// TIA Portal V16 export
// export: Created 2022-02-11T10:42:49.548867Z, ExportSetting WithDefaults, DisplayName Totally Integrated Automation Portal, DisplayVersion V16 Update 5, DisplayName TIA Portal Version Control Interface, DisplayVersion V16 Update 2, DisplayName TIA Portal Openness, DisplayVersion V16 Update 5, DisplayName STEP 7 Professional, DisplayVersion V16 Update 5, DisplayName STEP 7 Safety, DisplayVersion V16, DisplayName WinCC Professional, DisplayVersion V16 Update 5, DisplayName SIMATIC Visualization Architect, DisplayVersion V16
FUNCTION_BLOCK "fbObjEV_Aireacio"   // FB9102, LAD
{ S7_Optimized_Access := 'TRUE' }
VERSION : 0.1
// stored: AutoNumber false, IsIECCheckEnabled false, IsRetainMemResEnabled false, MemoryReserve 0, SetENOAutomatically false, UDAEnableTagReadback false
   VAR_INPUT
      eDP_PosTra : Bool := FALSE;   // Detector posicio valvula oberta
      eDP_PosAir : Bool := TRUE;   // Detector posicio valvula tancada
      aPosTra_Auto : Bool := FALSE;   // Ordre obrir EV en automatic
      psEnaAutoGrl : "boto";
      psEnaManualGrl : "boto";
      bCM_DirTra : Bool := TRUE;   // Condicions necesaries obrir valvula
      tAla_DirTra : Time := t#5s;   // Temps retard activacio alarma error obrir EV
      tAla_DirAir : Time := t#5s;   // Temps retard activacio alarma error tancar EV
      tAla_CM_DirTra : Time := t#3s;   // Temps retard activacio alarma condicions moviment
      psAnuConMov : Bool;
      psResetAlarma : Bool;
      mFirstScan : Bool;
      "Clock_0.5Hz" : Bool;
      bSysOk : Bool;
   END_VAR
   VAR_OUTPUT
      aPosTra : Bool;   // Sortida activacio EV
      be_DirTra : Bool;   // Bit estat EV oberta (Detectors + Sortida)
      be_DirAir : Bool;   // Bit estat EV tancada (Detectors + Sortida)
      al_CM_PosTra : Bool;   // Alarma condicions moviment obrir
      al_PosTra : Bool;   // Alarma obrir EV
      al_PosAir : Bool;   // Alarma tancar EV
      al_psEna : Bool;
   END_VAR
   VAR
      HMI { S7_SetPoint := 'True'} : "HMI_oEV";
      timAla_CM_DirTra : IEC_TIMER;   // Timer retard alarma condicions moviment
      timAla_DirTra : IEC_TIMER;   // Timer retard alarma obrirEV
      timAla_DirAir : IEC_TIMER;   // Timer retard alarma tancar EV
      mAuxTimer : Bool;   // Bit auxiliarInicialitzacio timers
      bLast_Reset : Bool;
   END_VAR
   VAR_TEMP
      ModeManual : Bool;
      ModeAutomatic : Bool;
      be_DirTra_Err : Bool;   // Error en validacio EV oberta. Sense retard per alarma.
      be_DirAir_Err : Bool;   // Error en validacio EV tancada. Sense retard per alarma.
      bCM_Ok : Bool;
      bErrorCM : Bool;   // Error CM. Si activem sortida i no es compleixen les CM. Sense retard
      aDirTraSenseTestCM : Bool;
      ResetAlarms : Bool;
   END_VAR
   VAR CONSTANT
      STATUS_OBJ_ERR : Int := 10;
      STATUS_OBJ_WARNING : Int := 11;
      STATUS_OBJ_ON : Int := 1;
      STATUS_OBJ_OFF : Int := 0;
      STATUS_OBJ_UNKNOWN : Int := -1;
   END_VAR
   VAR_TEMP   // added for the SCL form of the ladder/FBD networks
      _w1 : Bool;
   END_VAR
BEGIN

REGION Network 1 (SCL): Descripció
   // Motor amb guardamotor,confirmació i protecció.
END_REGION

REGION Network 2: Test habilitació mode manual. Desactivar si no tenim polsador manual o no tenim maniobra.
   // psEnaManualGrl : és el pulsador de manual de Appinfo. Si aquest està activar tots els objectes del cicle es troben en Mode Manual.
   // 
   // HMI.psEnaManual : és el pulsador de manual únic de l'objecte. Significa que la resta d'objectes es trobaràn en automàtic menys aquest.
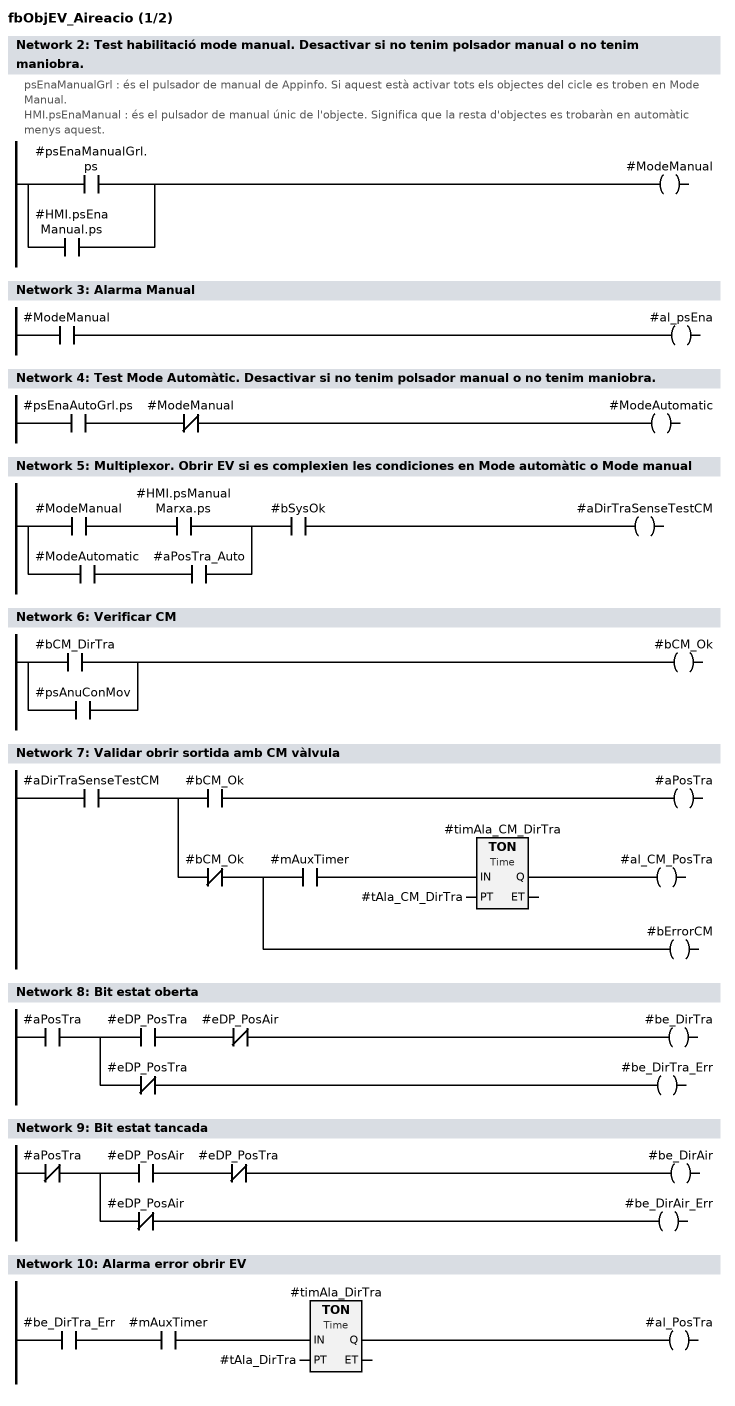
   RUNG wire#powerrail
      Contact( #psEnaManualGrl.ps )
      wire#w1
      Coil( #ModeManual )
   END_RUNG
   RUNG wire#powerrail
      Contact( #HMI.psEnaManual.ps )
   END_RUNG wire#w1
   // the same network as SCL:
   #ModeManual := #psEnaManualGrl.ps OR #HMI.psEnaManual.ps;
END_REGION

REGION Network 3: Alarma Manual
   RUNG wire#powerrail
      Contact( #ModeManual )
      Coil( #al_psEna )
   END_RUNG
   // the same network as SCL:
   #al_psEna := #ModeManual;
END_REGION

REGION Network 4: Test Mode Automàtic. Desactivar si no tenim polsador manual o no tenim maniobra.
   RUNG wire#powerrail
      Contact( #psEnaAutoGrl.ps )
      I_Contact( #ModeManual )
      Coil( #ModeAutomatic )
   END_RUNG
   // the same network as SCL:
   #ModeAutomatic := #psEnaAutoGrl.ps AND NOT #ModeManual;
END_REGION

REGION Network 5: Multiplexor. Obrir EV si es complexien les condiciones en Mode automàtic o Mode manual
   RUNG wire#powerrail
      Contact( #ModeManual )
      Contact( #HMI.psManualMarxa.ps )
      wire#w1
      Contact( #bSysOk )
      Coil( #aDirTraSenseTestCM )
   END_RUNG
   RUNG wire#powerrail
      Contact( #ModeAutomatic )
      Contact( #aPosTra_Auto )
   END_RUNG wire#w1
   // the same network as SCL:
   #aDirTraSenseTestCM := ((#ModeManual AND #HMI.psManualMarxa.ps) OR (#ModeAutomatic AND #aPosTra_Auto)) AND #bSysOk;
END_REGION

REGION Network 6: Verificar CM
   RUNG wire#powerrail
      Contact( #bCM_DirTra )
      wire#w1
      Coil( #bCM_Ok )
   END_RUNG
   RUNG wire#powerrail
      Contact( #psAnuConMov )
   END_RUNG wire#w1
   // the same network as SCL:
   #bCM_Ok := #bCM_DirTra OR #psAnuConMov;
END_REGION

REGION Network 7: Validar obrir sortida amb CM vàlvula
   RUNG wire#powerrail
      Contact( #aDirTraSenseTestCM )
      wire#w1
      Contact( #bCM_Ok )
      Coil( #aPosTra )
   END_RUNG
   RUNG wire#w1
      I_Contact( #bCM_Ok )
      wire#w2
      Contact( #mAuxTimer )
      { S7_Templates := "time_type := Time" } #timAla_CM_DirTra.TON(pt := #tAla_CM_DirTra, et =>)
      Coil( #al_CM_PosTra )
   END_RUNG
   RUNG wire#w2
      Coil( #bErrorCM )
   END_RUNG
   // the same network as SCL:
   #aPosTra := #aDirTraSenseTestCM AND #bCM_Ok;
   #_w1 := #aDirTraSenseTestCM AND NOT #bCM_Ok;
   #timAla_CM_DirTra.TON(IN := #_w1 AND #mAuxTimer, PT := #tAla_CM_DirTra);
   #al_CM_PosTra := #timAla_CM_DirTra.Q;
   #bErrorCM := #_w1;
END_REGION

REGION Network 8: Bit estat oberta
   RUNG wire#powerrail
      Contact( #aPosTra )
      wire#w1
      Contact( #eDP_PosTra )
      I_Contact( #eDP_PosAir )
      Coil( #be_DirTra )
   END_RUNG
   RUNG wire#w1
      I_Contact( #eDP_PosTra )
      Coil( #be_DirTra_Err )
   END_RUNG
   // the same network as SCL:
   #be_DirTra := #aPosTra AND #eDP_PosTra AND NOT #eDP_PosAir;
   #be_DirTra_Err := #aPosTra AND NOT #eDP_PosTra;
END_REGION

REGION Network 9: Bit estat tancada
   RUNG wire#powerrail
      I_Contact( #aPosTra )
      wire#w1
      Contact( #eDP_PosAir )
      I_Contact( #eDP_PosTra )
      Coil( #be_DirAir )
   END_RUNG
   RUNG wire#w1
      I_Contact( #eDP_PosAir )
      Coil( #be_DirAir_Err )
   END_RUNG
   // the same network as SCL:
   #be_DirAir := NOT #aPosTra AND #eDP_PosAir AND NOT #eDP_PosTra;
   #be_DirAir_Err := NOT #aPosTra AND NOT #eDP_PosAir;
END_REGION

REGION Network 10: Alarma error obrir EV
   RUNG wire#powerrail
      Contact( #be_DirTra_Err )
      Contact( #mAuxTimer )
      { S7_Templates := "time_type := Time" } #timAla_DirTra.TON(pt := #tAla_DirTra, et =>)
      Coil( #al_PosTra )
   END_RUNG
   // the same network as SCL:
   #timAla_DirTra.TON(IN := #be_DirTra_Err AND #mAuxTimer, PT := #tAla_DirTra);
   #al_PosTra := #timAla_DirTra.Q;
END_REGION

REGION Network 11: Alarma error tancar EV
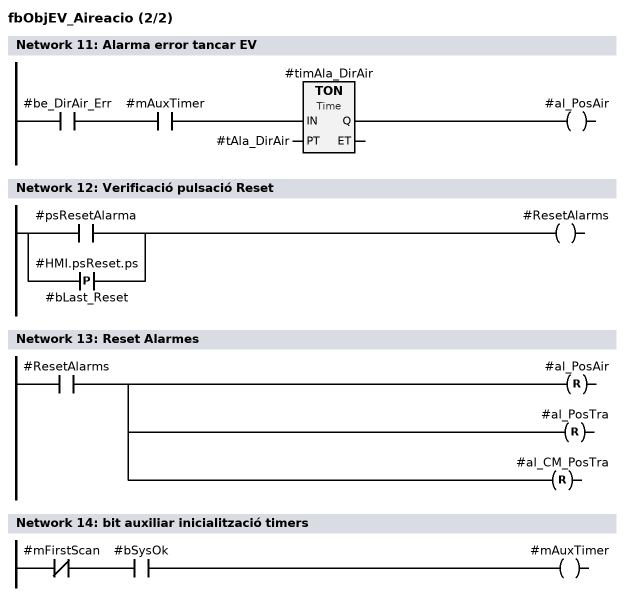
   RUNG wire#powerrail
      Contact( #be_DirAir_Err )
      Contact( #mAuxTimer )
      { S7_Templates := "time_type := Time" } #timAla_DirAir.TON(pt := #tAla_DirAir, et =>)
      Coil( #al_PosAir )
   END_RUNG
   // the same network as SCL:
   #timAla_DirAir.TON(IN := #be_DirAir_Err AND #mAuxTimer, PT := #tAla_DirAir);
   #al_PosAir := #timAla_DirAir.Q;
END_REGION

REGION Network 12: Verificació pulsació Reset
   RUNG wire#powerrail
      Contact( #psResetAlarma )
      wire#w1
      Coil( #ResetAlarms )
   END_RUNG
   RUNG wire#powerrail
      P_Contact(operand := #HMI.psReset.ps, bit := #bLast_Reset)
   END_RUNG wire#w1
   // the same network as SCL:
   #_w1 := #HMI.psReset.ps AND NOT #bLast_Reset;   // rising edge of #HMI.psReset.ps
   #bLast_Reset := #HMI.psReset.ps;
   #ResetAlarms := #psResetAlarma OR #_w1;
END_REGION

REGION Network 13: Reset Alarmes
   RUNG wire#powerrail
      Contact( #ResetAlarms )
      wire#w1
      R_Coil( #al_PosAir )
   END_RUNG
   RUNG wire#w1
      R_Coil( #al_PosTra )
   END_RUNG
   RUNG wire#w1
      R_Coil( #al_CM_PosTra )
   END_RUNG
   // the same network as SCL:
   IF #ResetAlarms THEN
       #al_PosAir := FALSE;
       #al_PosTra := FALSE;
       #al_CM_PosTra := FALSE;
   END_IF;
END_REGION

REGION Network 14: bit auxiliar inicialització timers
   RUNG wire#powerrail
      I_Contact( #mFirstScan )
      Contact( #bSysOk )
      Coil( #mAuxTimer )
   END_RUNG
   // the same network as SCL:
   #mAuxTimer := NOT #mFirstScan AND #bSysOk;
END_REGION

REGION Network 15 (SCL): HMI Estat EV
       IF (#al_PosTra OR #al_PosAir OR #al_CM_PosTra) THEN
           #HMI.iStatusDisplay := #STATUS_OBJ_ERR;                // Error = 10
           #HMI.bDisplayError := TRUE;
           #HMI.bDisplayWarning := FALSE;
           #HMI.bDisplayOk := FALSE;

       ELSIF (#be_DirTra_Err OR #be_DirAir_Err) THEN
           #HMI.iStatusDisplay := #STATUS_OBJ_WARNING;            // Warning = 11
           #HMI.bDisplayError := FALSE;
           #HMI.bDisplayWarning := TRUE;
           #HMI.bDisplayOk := FALSE;

       ELSIF #be_DirTra THEN
           #HMI.iStatusDisplay := #STATUS_OBJ_ON;                 // Bit estat Open Auto = 1
           #HMI.bDisplayError := FALSE;
           #HMI.bDisplayWarning := FALSE;
           #HMI.bDisplayOk := TRUE;

       ELSIF #be_DirAir THEN
           #HMI.iStatusDisplay := #STATUS_OBJ_OFF;               // Bit estat Close Automatic = 0
           #HMI.bDisplayError := FALSE;
           #HMI.bDisplayWarning := FALSE;
           #HMI.bDisplayOk := TRUE;

       ELSIF #aPosTra THEN
           IF #"Clock_0.5Hz" THEN
               #HMI.iStatusDisplay := #STATUS_OBJ_ON;
           ELSE
               #HMI.iStatusDisplay := #STATUS_OBJ_WARNING;
           END_IF;
           #HMI.bDisplayError := FALSE;
           #HMI.bDisplayWarning := FALSE;
           #HMI.bDisplayOk := TRUE;

       ELSE
           #HMI.iStatusDisplay := #STATUS_OBJ_UNKNOWN;            // Unknown = -1
           #HMI.bDisplayError := TRUE;
           #HMI.bDisplayWarning := FALSE;
           #HMI.bDisplayOk := FALSE;

       END_IF;

       #HMI.eON := #aPosTra;
       #HMI.eOFF := NOT #aPosTra;
       #HMI.error := #al_PosTra OR #al_PosAir;
       #HMI.confirmacio := #bSysOk;
END_REGION
END_FUNCTION_BLOCK
